// TIA Portal project "izpitni_projekt_v1_final" (V15.1)

(* hardware
DEVICE "S7-1200 station_1"  S7-1200 Station
   slot 0: "Rack_0"  S7-1200 Rack  Rack  V1.0
   slot 1: "PLC_1"  CPU 1214C DC/DC/DC  6ES7 214-1AG40-0XB0  V4.2
   slot 3: "AQ 1x12BIT_1"  AQ1 signal board  6ES7 232-4HA30-0XB0  V1.0
DEVICE "HMI_1"  TP900 Comfort
   slot 0: "HMI_1"  TP900 Comfort  6AV2 124-0JC01-0AX0  15.1.0.0
   slot 1: "HMI_RT_1"  TP900 Comfort  6AV2 124-0JC01-0AX0  15.1.0.0
   slot 5: "HMI_1.IE_CP_1"  PROFINET Interface  15.0.1.0
      slot 1: "PROFINET Interface_1"  PROFINET Interface
         slot 1: "Port_1"  Port
         slot 2: "Port_2"  Port
   slot 7: "HMI_1.MPI/DP_CP_1"  MPI/DP Interface  15.0.1.0
*)

// ===== PLC "PLC_1"  CPU 1214C DC/DC/DC =====
// protected blocks, not shown: "črna_škatlica"

VAR_GLOBAL   // PLC tag table "Default tag table"
   "Tag_1" AT %M0.0 : Bool;
   "Tag_2" AT %M0.1 : Bool;
   "Tag_3" AT %M0.2 : Bool;
   "Clock_Byte" AT %MB0 : Byte;
   "Clock_10Hz" AT %M0.0 : Bool;
   "Clock_5Hz" AT %M0.1 : Bool;
   "Clock_2.5Hz" AT %M0.2 : Bool;
   "Clock_2Hz" AT %M0.3 : Bool;
   "Clock_1.25Hz" AT %M0.4 : Bool;
   "Clock_1Hz" AT %M0.5 : Bool;
   "Clock_0.625Hz" AT %M0.6 : Bool;
   "Clock_0.5Hz" AT %M0.7 : Bool;
END_VAR

DATA_BLOCK "podatki_procesa"   // DB2
{ S7_Optimized_Access := 'TRUE' }
VERSION : 0.1
   VAR
      t_prek : Real := 0.05;   // čas prekinitve v s
      T_A : Real := 40.0;   // temperatura reagenta A
      T_B : Real := 20.0;   // temperatura reagenta B
      T_ok : Real := 20.0;   // temperatura okolice
      T_žel_max : Real := 85.0;   // maksimalna želena temperatura procesa
      deltaT_grad : Real := 1.0;   // gradient spremembe temperature (rampa v st. C/s)
      fi_A_max : Real := 500.0;   // pretok v ml/s
      fi_B_max : Real := 500.0;   // pretok v ml/s
      fi_OUT_max : Real := 500.0;   // pretok v ml/s
      t_heat : Real := 20.0;   // trajanje koraka 3 (vzdrževanje konst. temp.)
      ro_A : Real := 0.81;
      ro_B : Real := 1.0;
      "%_A" : Real := 0.96;
      V_žel : Real;
      "%_žel" : Real;
      T_Žel : Real;
      V_A : Real;
      V_B : Real;
      Grelec1_power : DInt := 5000;
      Grelec2_power : DInt := 20000;
      Grelec3_power : DInt := 70000;
      Spec_Toplota_Voda : Int := 4182;
      Spec_Toplota_Alkohol : Int := 2440;
      Toplotne_Izgube_Koeficient : Real := -2.409683;   // Izmerjene Toplotne izgube 289.0, 267.5585, trial & error -2.409683
      Toplotne_Izgube_Voda : Real := 400.0;   // Somehow so Toplotne izgube povezane z % razkuzila xd
   END_VAR
BEGIN
END_DATA_BLOCK

DATA_BLOCK "spremenljivke"   // DB3
{ S7_Optimized_Access := 'TRUE' }
VERSION : 0.1
   VAR
      reset_DB : Bool;   // tipka reset
      glavno_stikalo_DB : Bool := true;
      zasilni_izklop_DB : Bool;
      avtomatično : Bool := true;
      Ventil_voda : Bool;
      Ventil_alkohol : Bool;
      Ventil_out : Bool;
      Mešalo : Bool;
      Korak1 : Bool;
      Korak2 : Bool;
      Korak3 : Bool;
      Korak4 : Bool;
      Grelec1 : Bool;
      Grelec2 : Bool;
      Grelec3 : Bool;
      Volumen : Real;
      Temperatura : Real;
      prejsna_temp : Real;
      Temp_gradient : Real;
      "%_trenutni" : Real;
      L_zg : Bool;
      L_sp : Bool;
      Pretok_alkohol_mapped : Real;
      Pretok_alkohol : Real;
      Pretok_Voda_mapped : Real;
      Pretok_Voda : Real;
      RMSE_T : Real;
      Error : Word;
   END_VAR
BEGIN
END_DATA_BLOCK

DATA_BLOCK "Korak1_DB"   // DB4
{ S7_Optimized_Access := 'TRUE' }
VERSION : 0.1
// stored: InstanceOfName Korak1
"Korak1"
BEGIN
END_DATA_BLOCK

DATA_BLOCK "Korak3_DB"   // DB5
{ S7_Optimized_Access := 'TRUE' }
VERSION : 0.1
// stored: InstanceOfName Korak3
"Korak3"
BEGIN
END_DATA_BLOCK

DATA_BLOCK "Korak2_DB"   // DB7
{ S7_Optimized_Access := 'TRUE' }
VERSION : 0.1
// stored: InstanceOfName Korak2
"Korak2"
BEGIN
END_DATA_BLOCK

FUNCTION_BLOCK "Korak1"   // FB2, LAD
{ S7_Optimized_Access := 'TRUE' }
VERSION : 0.1
   VAR_INPUT
      reset : Bool;
      "counter" : DInt;
   END_VAR
   VAR_OUTPUT
      finnished : Bool;
   END_VAR
   VAR
      interrupts_count : DInt;
   END_VAR
   VAR_TEMP
      "cas ventil voda" : Time;
      interrupts_voda : Int;
      "cas ventil alkohol" : Time;
      interrupts_alkohol : Int;
   END_VAR
   VAR_TEMP   // added for the SCL form of the ladder/FBD networks
      _w1 : Bool;
      _w2 : Bool;
   END_VAR
BEGIN

REGION Network 1
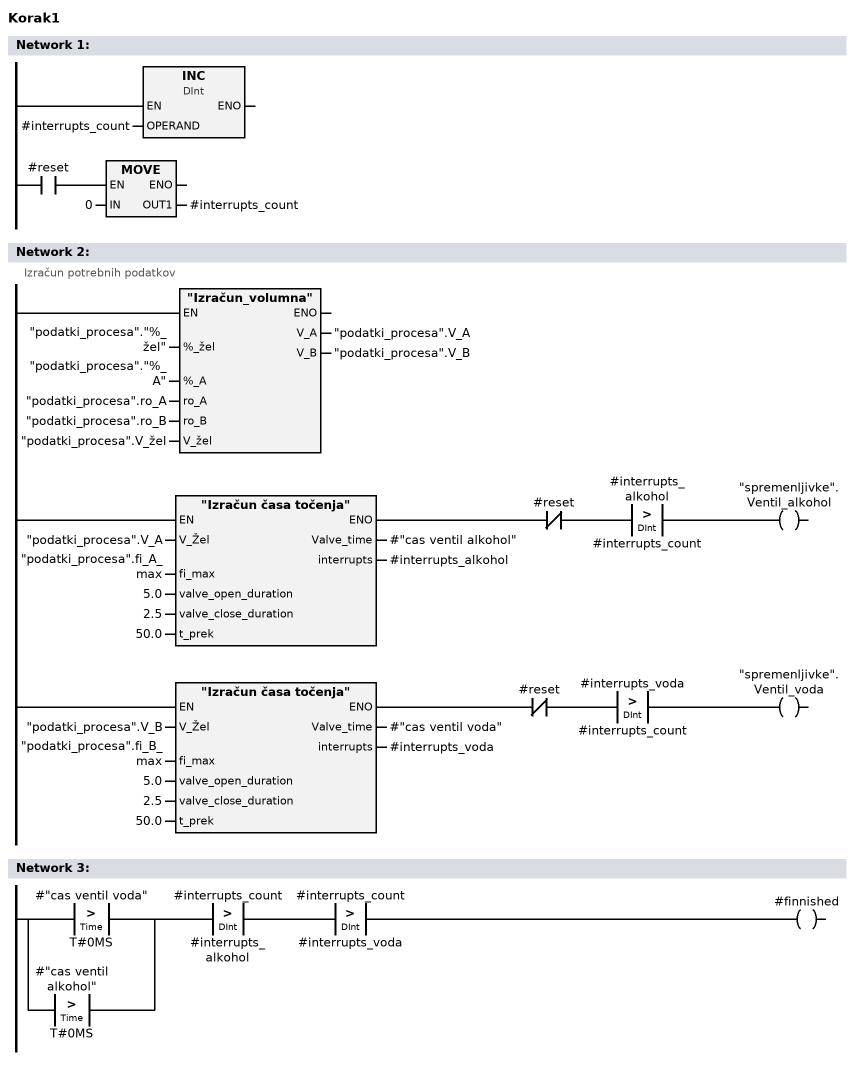
   RUNG wire#powerrail
      { S7_Templates := "DestType := DInt" } Inc( #interrupts_count )
   END_RUNG
   RUNG wire#powerrail
      Contact( #reset )
      Move(in := 0, out1 => #interrupts_count)
   END_RUNG
   // the same network as SCL:
   #interrupts_count := #interrupts_count + 1;
   IF #reset THEN #interrupts_count := 0; END_IF;
END_REGION

REGION Network 2
   // Izračun potrebnih podatkov
   RUNG wire#powerrail
      "Izračun_volumna"("%_žel" := "podatki_procesa"."%_žel", "%_A" := "podatki_procesa"."%_A", ro_A := "podatki_procesa".ro_A, ro_B := "podatki_procesa".ro_B, V_žel := "podatki_procesa".V_žel, V_A => "podatki_procesa".V_A, V_B => "podatki_procesa".V_B)
   END_RUNG
   RUNG wire#powerrail
      "Izračun časa točenja"(V_Žel := "podatki_procesa".V_A, fi_max := "podatki_procesa".fi_A_max, valve_open_duration := 5.0, valve_close_duration := 2.5, t_prek := 50.0, Valve_time => #"cas ventil alkohol", interrupts => #interrupts_alkohol)
      I_Contact( #reset )
      { S7_Templates := "SrcType := DInt" } GT_Contact(in1 := #interrupts_alkohol, in2 := #interrupts_count)
      Coil( "spremenljivke".Ventil_alkohol )
   END_RUNG
   RUNG wire#powerrail
      "Izračun časa točenja"(V_Žel := "podatki_procesa".V_B, fi_max := "podatki_procesa".fi_B_max, valve_open_duration := 5.0, valve_close_duration := 2.5, t_prek := 50.0, Valve_time => #"cas ventil voda", interrupts => #interrupts_voda)
      I_Contact( #reset )
      { S7_Templates := "SrcType := DInt" } GT_Contact(in1 := #interrupts_voda, in2 := #interrupts_count)
      Coil( "spremenljivke".Ventil_voda )
   END_RUNG
   // the same network as SCL:
   "Izračun_volumna"("%_žel" := "podatki_procesa"."%_žel",
                     "%_A" := "podatki_procesa"."%_A",
                     ro_A := "podatki_procesa".ro_A,
                     ro_B := "podatki_procesa".ro_B,
                     V_žel := "podatki_procesa".V_žel,
                     V_A => "podatki_procesa".V_A,
                     V_B => "podatki_procesa".V_B);
   "Izračun časa točenja"(V_Žel := "podatki_procesa".V_A,
                          fi_max := "podatki_procesa".fi_A_max,
                          valve_open_duration := 5.0,
                          valve_close_duration := 2.5,
                          t_prek := 50.0,
                          Valve_time => #"cas ventil alkohol",
                          interrupts => #interrupts_alkohol,
                          ENO => #_w1);
   "spremenljivke".Ventil_alkohol := #_w1 AND NOT #reset AND (#interrupts_alkohol > #interrupts_count);
   "Izračun časa točenja"(V_Žel := "podatki_procesa".V_B,
                          fi_max := "podatki_procesa".fi_B_max,
                          valve_open_duration := 5.0,
                          valve_close_duration := 2.5,
                          t_prek := 50.0,
                          Valve_time => #"cas ventil voda",
                          interrupts => #interrupts_voda,
                          ENO => #_w2);
   "spremenljivke".Ventil_voda := #_w2 AND NOT #reset AND (#interrupts_voda > #interrupts_count);
END_REGION

REGION Network 3
   RUNG wire#powerrail
      { S7_Templates := "SrcType := Time" } GT_Contact(in1 := #"cas ventil voda", in2 := T#0MS)
      wire#w1
      { S7_Templates := "SrcType := DInt" } GT_Contact(in1 := #interrupts_count, in2 := #interrupts_alkohol)
      { S7_Templates := "SrcType := DInt" } GT_Contact(in1 := #interrupts_count, in2 := #interrupts_voda)
      Coil( #finnished )
   END_RUNG
   RUNG wire#powerrail
      { S7_Templates := "SrcType := Time" } GT_Contact(in1 := #"cas ventil alkohol", in2 := T#0MS)
   END_RUNG wire#w1
   // the same network as SCL:
   #finnished := ((#"cas ventil voda" > T#0MS) OR (#"cas ventil alkohol" > T#0MS)) AND (#interrupts_count > #interrupts_alkohol) AND (#interrupts_count > #interrupts_voda);
END_REGION
END_FUNCTION_BLOCK

FUNCTION_BLOCK "Korak2"   // FB3, LAD
{ S7_Optimized_Access := 'TRUE' }
VERSION : 0.1
   VAR_INPUT
      reset : Bool;
   END_VAR
   VAR_OUTPUT
      finnished : Bool;
   END_VAR
   VAR
      interrupts_count : DInt;
      Upravljaj_grelce_Instance : "Upravljaj_grelce";
      Upravljaj_grelce_Instance_1 : "Upravljaj_grelce";
   END_VAR
   VAR_TEMP
      "Energija/K_Total" : Real;
      "Energija/K_Alkohol" : Real;
      "Energija/K_Voda_Alko" : Real;
      "Energija/K_Voda" : Real;
      "%_vode_v_alko" : Real;
      Toplotne_izbuge : Real;
      Potrebna_energija : Real;
      ElapsedTime : Time;
   END_VAR
BEGIN

REGION Network 1
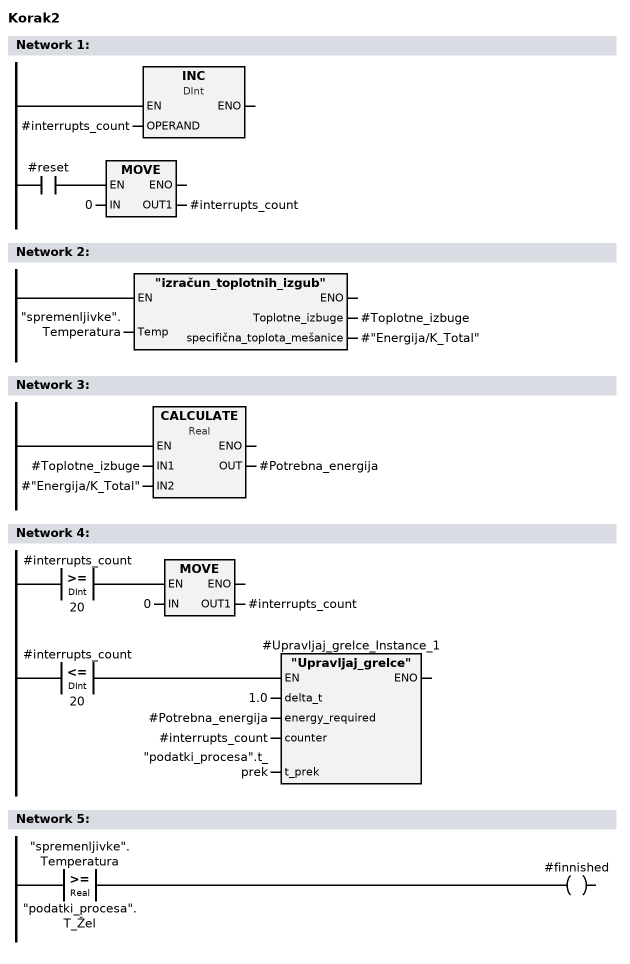
   RUNG wire#powerrail
      { S7_Templates := "DestType := DInt" } Inc( #interrupts_count )
   END_RUNG
   RUNG wire#powerrail
      Contact( #reset )
      Move(in := 0, out1 => #interrupts_count)
   END_RUNG
   // the same network as SCL:
   #interrupts_count := #interrupts_count + 1;
   IF #reset THEN #interrupts_count := 0; END_IF;
END_REGION

REGION Network 2
   RUNG wire#powerrail
      "izračun_toplotnih_izgub"(Temp := "spremenljivke".Temperatura, Toplotne_izbuge => #Toplotne_izbuge, specifična_toplota_mešanice => #"Energija/K_Total")
   END_RUNG
   // the same network as SCL:
   "izračun_toplotnih_izgub"(Temp := "spremenljivke".Temperatura,
                           Toplotne_izbuge => #Toplotne_izbuge,
                           specifična_toplota_mešanice => #"Energija/K_Total");
END_REGION

REGION Network 3
   RUNG wire#powerrail
      { S7_Templates := "SrcType := Real"; S7_Expression := "(IN1 + IN2)" } Calculate(in1 := #Toplotne_izbuge, in2 := #"Energija/K_Total", out => #Potrebna_energija)
   END_RUNG
   // the same network as SCL:
   #Potrebna_energija := (#Toplotne_izbuge + #"Energija/K_Total");
END_REGION

REGION Network 4
   RUNG wire#powerrail
      { S7_Templates := "SrcType := DInt" } GE_Contact(in1 := #interrupts_count, in2 := 20)
      Move(in := 0, out1 => #interrupts_count)
   END_RUNG
   RUNG wire#powerrail
      { S7_Templates := "SrcType := DInt" } LE_Contact(in1 := #interrupts_count, in2 := 20)
      #Upravljaj_grelce_Instance_1(delta_t := 1.0, energy_required := #Potrebna_energija, "counter" := #interrupts_count, t_prek := "podatki_procesa".t_prek)
   END_RUNG
   // the same network as SCL:
   IF #interrupts_count >= 20 THEN #interrupts_count := 0; END_IF;
   IF #interrupts_count <= 20 THEN
       #Upravljaj_grelce_Instance_1(delta_t := 1.0,   // "Upravljaj_grelce"
                               energy_required := #Potrebna_energija,
                               "counter" := #interrupts_count,
                               t_prek := "podatki_procesa".t_prek);
   END_IF;
END_REGION

REGION Network 5
   RUNG wire#powerrail
      { S7_Templates := "SrcType := Real" } GE_Contact(in1 := "spremenljivke".Temperatura, in2 := "podatki_procesa".T_Žel)
      Coil( #finnished )
   END_RUNG
   // the same network as SCL:
   #finnished := "spremenljivke".Temperatura >= "podatki_procesa".T_Žel;
END_REGION
END_FUNCTION_BLOCK

FUNCTION_BLOCK "Upravljaj_grelce"   // FB4, LAD
{ S7_Optimized_Access := 'TRUE' }
VERSION : 0.1
   VAR_INPUT
      delta_t : Real;
      energy_required : LReal;
      "counter" : Int;
      t_prek : Real;
   END_VAR
   VAR
      energy_delivered : LReal;
      energy_missing : Real;
   END_VAR
   VAR_TEMP
      power : Real;
      energy_heater1 : Real;
      energy_heater2 : Real;
      energy_heater3 : Real;
   END_VAR
   VAR_TEMP   // added for the SCL form of the ladder/FBD networks
      _w1 : Bool;
   END_VAR
BEGIN

REGION Network 1
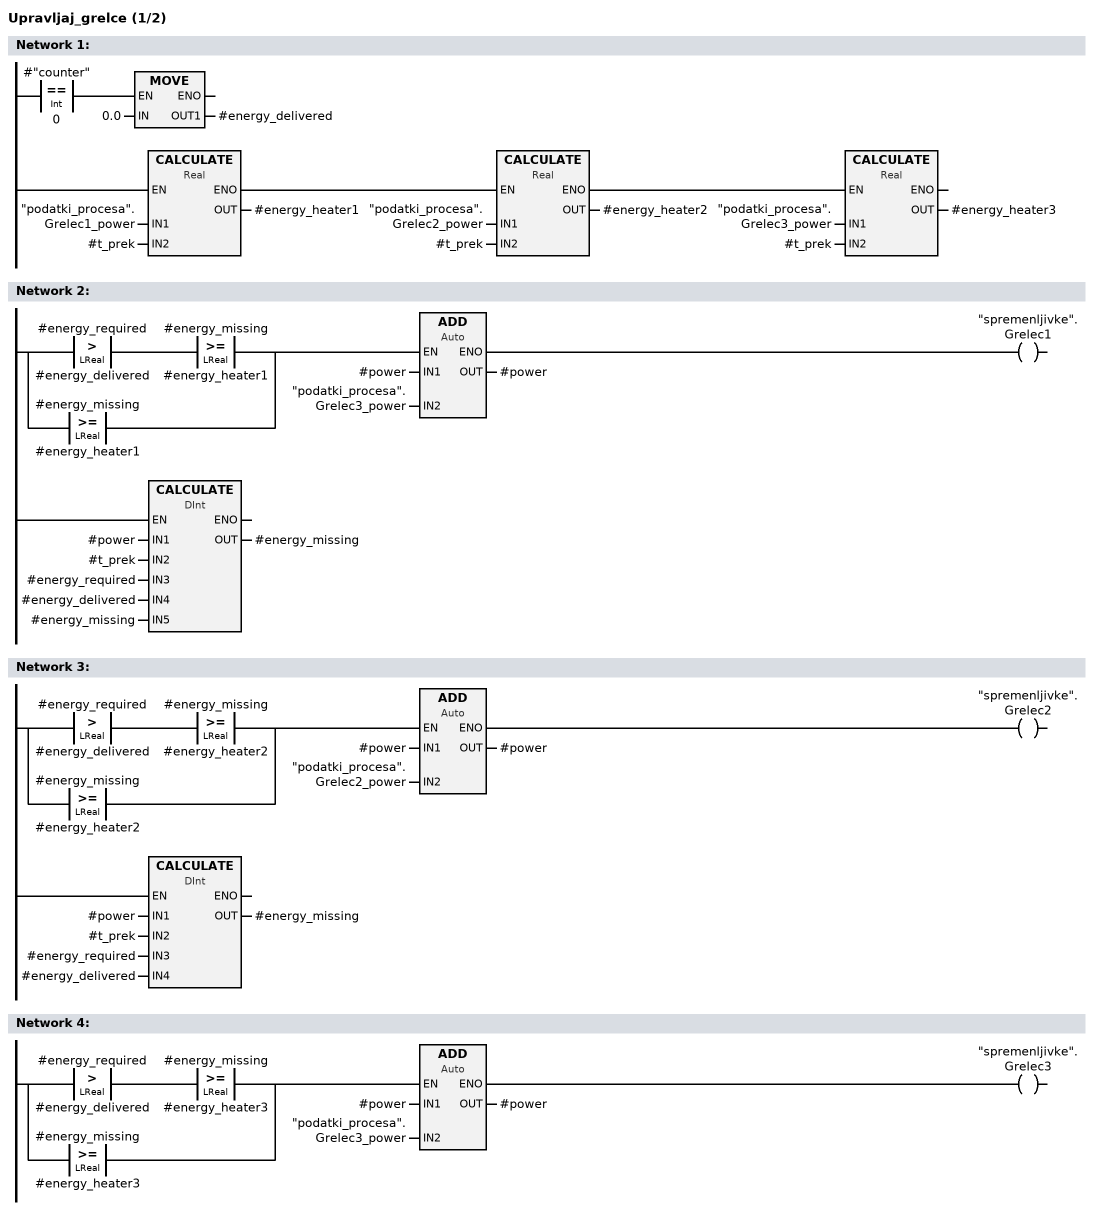
   RUNG wire#powerrail
      { S7_Templates := "SrcType := Int" } EQ_Contact(in1 := #"counter", in2 := 0)
      Move(in := 0.0, out1 => #energy_delivered)
   END_RUNG
   RUNG wire#powerrail
      { S7_Templates := "SrcType := Real"; S7_Expression := "IN1*IN2" } Calculate(in1 := "podatki_procesa".Grelec1_power, in2 := #t_prek, out => #energy_heater1)
      { S7_Templates := "SrcType := Real"; S7_Expression := "IN1*IN2" } Calculate(in1 := "podatki_procesa".Grelec2_power, in2 := #t_prek, out => #energy_heater2)
      { S7_Templates := "SrcType := Real"; S7_Expression := "IN1*IN2" } Calculate(in1 := "podatki_procesa".Grelec3_power, in2 := #t_prek, out => #energy_heater3)
   END_RUNG
   // the same network as SCL:
   IF #"counter" = 0 THEN #energy_delivered := 0.0; END_IF;
   #energy_heater1 := "podatki_procesa".Grelec1_power*#t_prek;
   #energy_heater2 := "podatki_procesa".Grelec2_power*#t_prek;
   #energy_heater3 := "podatki_procesa".Grelec3_power*#t_prek;
END_REGION

REGION Network 2
   RUNG wire#powerrail
      { S7_Templates := "SrcType := LReal" } GT_Contact(in1 := #energy_required, in2 := #energy_delivered)
      { S7_Templates := "SrcType := LReal" } GE_Contact(in1 := #energy_missing, in2 := #energy_heater1)
      wire#w1
      Add(in1 := #power, in2 := "podatki_procesa".Grelec3_power, out => #power)
      Coil( "spremenljivke".Grelec1 )
   END_RUNG
   RUNG wire#powerrail
      { S7_Templates := "SrcType := LReal" } GE_Contact(in1 := #energy_missing, in2 := #energy_heater1)
   END_RUNG wire#w1
   RUNG wire#powerrail
      { S7_Templates := "SrcType := DInt"; S7_Expression := "(IN3-IN4-IN1*IN2 )+ IN5" } Calculate(in1 := #power, in2 := #t_prek, in3 := #energy_required, in4 := #energy_delivered, in5 := #energy_missing, out => #energy_missing)
   END_RUNG
   // the same network as SCL:
   #_w1 := ((#energy_required > #energy_delivered) AND (#energy_missing >= #energy_heater1)) OR (#energy_missing >= #energy_heater1);
   IF #_w1 THEN #power := #power + "podatki_procesa".Grelec3_power; END_IF;
   "spremenljivke".Grelec1 := #_w1;
   #energy_missing := (#energy_required-#energy_delivered-#power*#t_prek )+ #energy_missing;
END_REGION

REGION Network 3
   RUNG wire#powerrail
      { S7_Templates := "SrcType := LReal" } GT_Contact(in1 := #energy_required, in2 := #energy_delivered)
      { S7_Templates := "SrcType := LReal" } GE_Contact(in1 := #energy_missing, in2 := #energy_heater2)
      wire#w1
      Add(in1 := #power, in2 := "podatki_procesa".Grelec2_power, out => #power)
      Coil( "spremenljivke".Grelec2 )
   END_RUNG
   RUNG wire#powerrail
      { S7_Templates := "SrcType := LReal" } GE_Contact(in1 := #energy_missing, in2 := #energy_heater2)
   END_RUNG wire#w1
   RUNG wire#powerrail
      { S7_Templates := "SrcType := DInt"; S7_Expression := "IN3-IN4-IN1*IN2" } Calculate(in1 := #power, in2 := #t_prek, in3 := #energy_required, in4 := #energy_delivered, out => #energy_missing)
   END_RUNG
   // the same network as SCL:
   #_w1 := ((#energy_required > #energy_delivered) AND (#energy_missing >= #energy_heater2)) OR (#energy_missing >= #energy_heater2);
   IF #_w1 THEN #power := #power + "podatki_procesa".Grelec2_power; END_IF;
   "spremenljivke".Grelec2 := #_w1;
   #energy_missing := #energy_required-#energy_delivered-#power*#t_prek;
END_REGION

REGION Network 4
   RUNG wire#powerrail
      { S7_Templates := "SrcType := LReal" } GT_Contact(in1 := #energy_required, in2 := #energy_delivered)
      { S7_Templates := "SrcType := LReal" } GE_Contact(in1 := #energy_missing, in2 := #energy_heater3)
      wire#w1
      Add(in1 := #power, in2 := "podatki_procesa".Grelec3_power, out => #power)
      Coil( "spremenljivke".Grelec3 )
   END_RUNG
   RUNG wire#powerrail
      { S7_Templates := "SrcType := LReal" } GE_Contact(in1 := #energy_missing, in2 := #energy_heater3)
   END_RUNG wire#w1
   // the same network as SCL:
   #_w1 := ((#energy_required > #energy_delivered) AND (#energy_missing >= #energy_heater3)) OR (#energy_missing >= #energy_heater3);
   IF #_w1 THEN #power := #power + "podatki_procesa".Grelec3_power; END_IF;
   "spremenljivke".Grelec3 := #_w1;
END_REGION

REGION Network 5
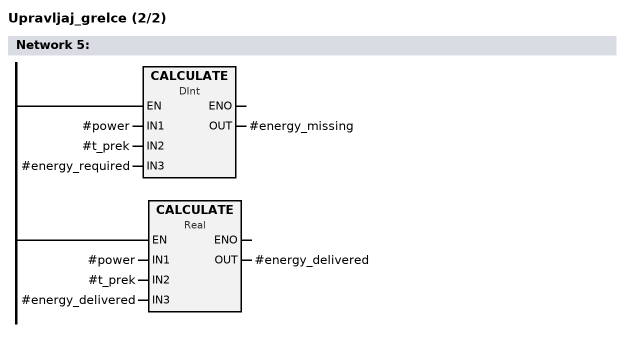
   RUNG wire#powerrail
      { S7_Templates := "SrcType := DInt"; S7_Expression := "IN3-IN1*IN2" } Calculate(in1 := #power, in2 := #t_prek, in3 := #energy_required, out => #energy_missing)
   END_RUNG
   RUNG wire#powerrail
      { S7_Templates := "SrcType := Real"; S7_Expression := "IN3 + IN1 * IN2" } Calculate(in1 := #power, in2 := #t_prek, in3 := #energy_delivered, out => #energy_delivered)
   END_RUNG
   // the same network as SCL:
   #energy_missing := #energy_required-#power*#t_prek;
   #energy_delivered := #energy_delivered + #power * #t_prek;
END_REGION
END_FUNCTION_BLOCK

FUNCTION_BLOCK "Korak3"   // FB5, LAD
{ S7_Optimized_Access := 'TRUE' }
VERSION : 0.1
   VAR_INPUT
      reset : Bool;
   END_VAR
   VAR_OUTPUT
      finnished_1 : Bool;
   END_VAR
   VAR
      Upravljaj_grelce_Instance : "Upravljaj_grelce";
      interrupts_count : DInt;
   END_VAR
   VAR_TEMP
      "toplotne izgube" : Real;
      "specificna toplota" : Real;
   END_VAR
BEGIN

REGION Network 1
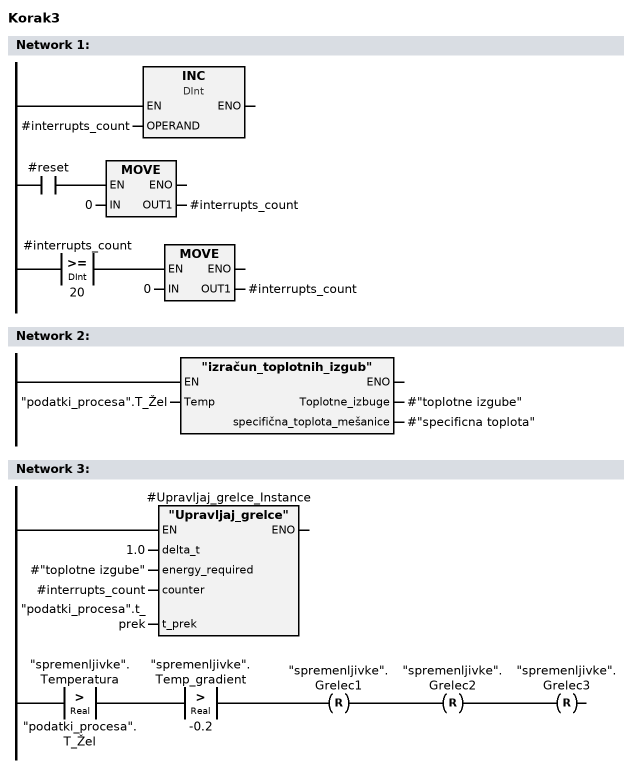
   RUNG wire#powerrail
      { S7_Templates := "DestType := DInt" } Inc( #interrupts_count )
   END_RUNG
   RUNG wire#powerrail
      Contact( #reset )
      Move(in := 0, out1 => #interrupts_count)
   END_RUNG
   RUNG wire#powerrail
      { S7_Templates := "SrcType := DInt" } GE_Contact(in1 := #interrupts_count, in2 := 20)
      Move(in := 0, out1 => #interrupts_count)
   END_RUNG
   // the same network as SCL:
   #interrupts_count := #interrupts_count + 1;
   IF #reset THEN #interrupts_count := 0; END_IF;
   IF #interrupts_count >= 20 THEN #interrupts_count := 0; END_IF;
END_REGION

REGION Network 2
   RUNG wire#powerrail
      "izračun_toplotnih_izgub"(Temp := "podatki_procesa".T_Žel, Toplotne_izbuge => #"toplotne izgube", specifična_toplota_mešanice => #"specificna toplota")
   END_RUNG
   // the same network as SCL:
   "izračun_toplotnih_izgub"(Temp := "podatki_procesa".T_Žel,
                           Toplotne_izbuge => #"toplotne izgube",
                           specifična_toplota_mešanice => #"specificna toplota");
END_REGION

REGION Network 3
   RUNG wire#powerrail
      #Upravljaj_grelce_Instance(delta_t := 1.0, energy_required := #"toplotne izgube", "counter" := #interrupts_count, t_prek := "podatki_procesa".t_prek)
   END_RUNG
   RUNG wire#powerrail
      { S7_Templates := "SrcType := Real" } GT_Contact(in1 := "spremenljivke".Temperatura, in2 := "podatki_procesa".T_Žel)
      { S7_Templates := "SrcType := Real" } GT_Contact(in1 := "spremenljivke".Temp_gradient, in2 := -0.2)
      R_Coil( "spremenljivke".Grelec1 )
      R_Coil( "spremenljivke".Grelec2 )
      R_Coil( "spremenljivke".Grelec3 )
   END_RUNG
   // the same network as SCL:
   #Upravljaj_grelce_Instance(delta_t := 1.0,   // "Upravljaj_grelce"
                           energy_required := #"toplotne izgube",
                           "counter" := #interrupts_count,
                           t_prek := "podatki_procesa".t_prek);
   IF ("spremenljivke".Temperatura > "podatki_procesa".T_Žel) AND ("spremenljivke".Temp_gradient > (-0.2)) THEN
       "spremenljivke".Grelec1 := FALSE;
       "spremenljivke".Grelec2 := FALSE;
       "spremenljivke".Grelec3 := FALSE;
   END_IF;
END_REGION
END_FUNCTION_BLOCK

FUNCTION "map_Flow_Sensor" : Void   // FC1, LAD
{ S7_Optimized_Access := 'TRUE' }
VERSION : 0.1
   VAR_INPUT
      input_value : Real;
      max_value : Real;
   END_VAR
   VAR_OUTPUT
      output_value : Real;
   END_VAR
   VAR_TEMP
      norm_Value : Real;
   END_VAR
BEGIN

REGION Network 1
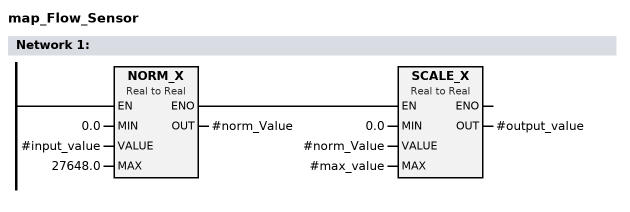
   RUNG wire#powerrail
      { S7_Templates := "[SrcType := Real, DestType := Real]" } Normalize(min := 0.0, value := #input_value, max := 27648.0, out => #norm_Value)
      { S7_Templates := "[SrcType := Real, DestType := Real]" } Scale(min := 0.0, value := #norm_Value, max := #max_value, out => #output_value)
   END_RUNG
   // the same network as SCL:
   #norm_Value := NORM_X(MIN := 0.0, VALUE := #input_value, MAX := 27648.0);
   #output_value := SCALE_X(MIN := 0.0, VALUE := #norm_Value, MAX := #max_value);
END_REGION
END_FUNCTION

FUNCTION "Izračun_volumna" : Void   // FC2, LAD
{ S7_Optimized_Access := 'TRUE' }
VERSION : 0.1
   VAR_INPUT
      "%_žel" : Real;
      "%_A" : Real;
      ro_A : Real;
      ro_B : Real;
      V_žel : Real;
   END_VAR
   VAR_OUTPUT
      V_A : Real;
      V_B : Real;
   END_VAR
   VAR_TEMP
      "V_B/V_A" : Real;   // Razmerje volumen Vode / Volumen Alkohola
   END_VAR
BEGIN

REGION Network 1
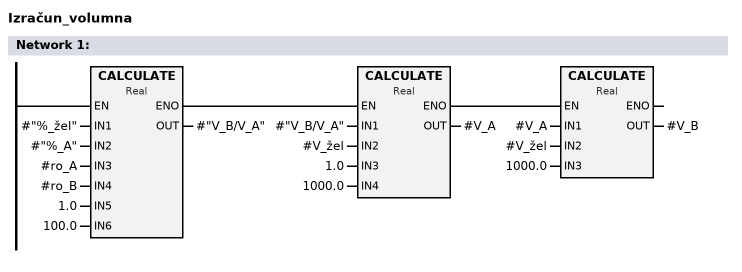
   RUNG wire#powerrail
      { S7_Templates := "SrcType := Real"; S7_Expression := "((IN3 * IN2)/((IN1/IN6) * IN4)) - ((IN3*(IN5-IN2))/IN4) -((IN3 * IN2)/(IN4))" } Calculate(in1 := #"%_žel", in2 := #"%_A", in3 := #ro_A, in4 := #ro_B, in5 := 1.0, in6 := 100.0, out => #"V_B/V_A")
      { S7_Templates := "SrcType := Real"; S7_Expression := "(IN2*IN4)/(IN3+IN1)" } Calculate(in1 := #"V_B/V_A", in2 := #V_žel, in3 := 1.0, in4 := 1000.0, out => #V_A)
      { S7_Templates := "SrcType := Real"; S7_Expression := "(IN2 * IN3) - IN1" } Calculate(in1 := #V_A, in2 := #V_žel, in3 := 1000.0, out => #V_B)
   END_RUNG
   // the same network as SCL:
   #"V_B/V_A" := ((#ro_A * #"%_A")/((#"%_žel"/100.0) * #ro_B)) - ((#ro_A*(1.0-#"%_A"))/#ro_B) -((#ro_A * #"%_A")/(#ro_B));
   #V_A := (#V_žel*1000.0)/(1.0+#"V_B/V_A");
   #V_B := (#V_žel * 1000.0) - #V_A;
END_REGION
END_FUNCTION

FUNCTION "izračun_toplotnih_izgub" : Void   // FC3, LAD
{ S7_Optimized_Access := 'TRUE' }
VERSION : 0.1
   VAR_INPUT
      Temp : Real;
   END_VAR
   VAR_OUTPUT
      Toplotne_izbuge : Real;
      specifična_toplota_mešanice : Real;
   END_VAR
   VAR_TEMP
      "Energija/K_Alkohol" : Real;
      "Energija/K_Voda_Alko" : Real;
      "Energija/K_Voda" : Real;
      "%_vode_v_alko" : Real;
      Potrebna_energija : Real;
   END_VAR
   VAR_TEMP   // added for the SCL form of the ladder/FBD networks
      _w1 : Bool;
   END_VAR
BEGIN

REGION Network 1
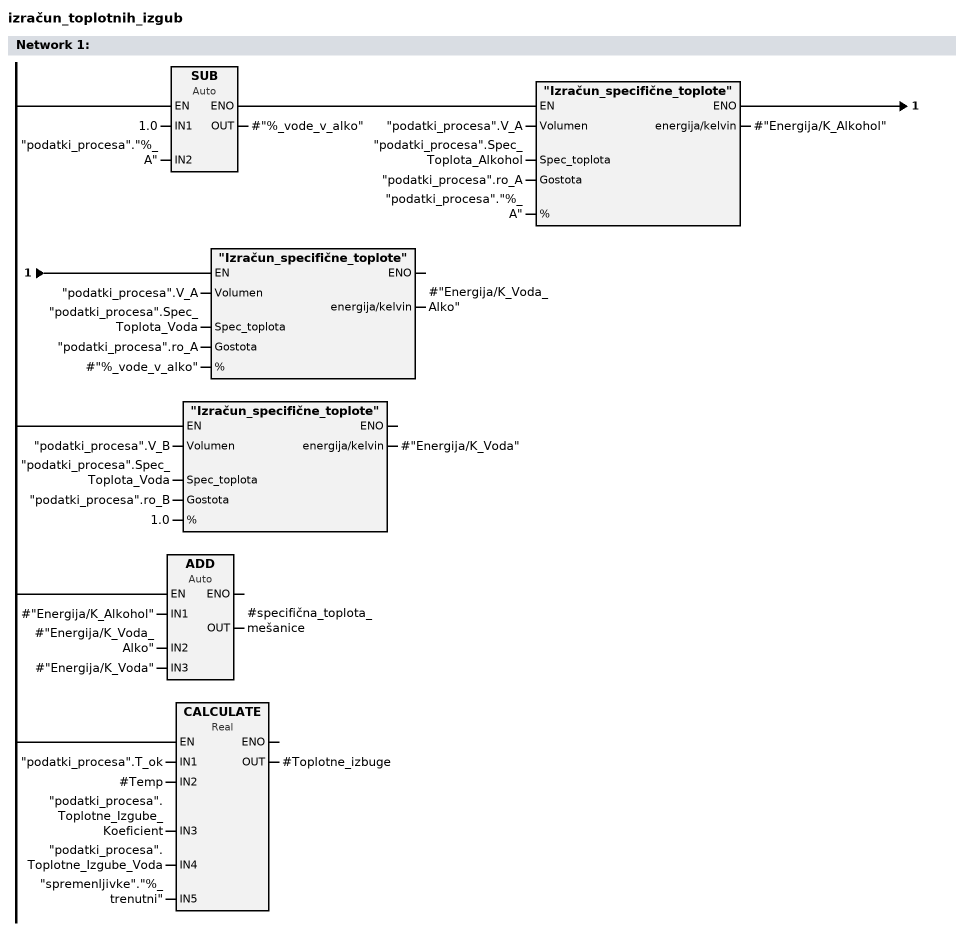
   RUNG wire#powerrail
      Sub(in1 := 1.0, in2 := "podatki_procesa"."%_A", out => #"%_vode_v_alko")
      "Izračun_specifične_toplote"(Volumen := "podatki_procesa".V_A, Spec_toplota := "podatki_procesa".Spec_Toplota_Alkohol, Gostota := "podatki_procesa".ro_A, "%" := "podatki_procesa"."%_A", "energija/kelvin" => #"Energija/K_Alkohol")
      "Izračun_specifične_toplote"(Volumen := "podatki_procesa".V_A, Spec_toplota := "podatki_procesa".Spec_Toplota_Voda, Gostota := "podatki_procesa".ro_A, "%" := #"%_vode_v_alko", "energija/kelvin" => #"Energija/K_Voda_Alko")
   END_RUNG
   RUNG wire#powerrail
      "Izračun_specifične_toplote"(Volumen := "podatki_procesa".V_B, Spec_toplota := "podatki_procesa".Spec_Toplota_Voda, Gostota := "podatki_procesa".ro_B, "%" := 1.0, "energija/kelvin" => #"Energija/K_Voda")
   END_RUNG
   RUNG wire#powerrail
      Add(in1 := #"Energija/K_Alkohol", in2 := #"Energija/K_Voda_Alko", in3 := #"Energija/K_Voda", out => #specifična_toplota_mešanice)
   END_RUNG
   RUNG wire#powerrail
      { S7_Templates := "SrcType := Real"; S7_Expression := "(IN3*IN5 + IN4) * (IN2-IN1)" } Calculate(in1 := "podatki_procesa".T_ok, in2 := #Temp, in3 := "podatki_procesa".Toplotne_Izgube_Koeficient, in4 := "podatki_procesa".Toplotne_Izgube_Voda, in5 := "spremenljivke"."%_trenutni", out => #Toplotne_izbuge)
   END_RUNG
   // the same network as SCL:
   #"%_vode_v_alko" := 1.0 - "podatki_procesa"."%_A";
   "Izračun_specifične_toplote"(Volumen := "podatki_procesa".V_A,
                           Spec_toplota := "podatki_procesa".Spec_Toplota_Alkohol,
                           Gostota := "podatki_procesa".ro_A,
                           "%" := "podatki_procesa"."%_A",
                           "energija/kelvin" => #"Energija/K_Alkohol",
                           ENO => #_w1);
   IF #_w1 THEN
       "Izračun_specifične_toplote"(Volumen := "podatki_procesa".V_A,
                               Spec_toplota := "podatki_procesa".Spec_Toplota_Voda,
                               Gostota := "podatki_procesa".ro_A,
                               "%" := #"%_vode_v_alko",
                               "energija/kelvin" => #"Energija/K_Voda_Alko");
   END_IF;
   "Izračun_specifične_toplote"(Volumen := "podatki_procesa".V_B,
                           Spec_toplota := "podatki_procesa".Spec_Toplota_Voda,
                           Gostota := "podatki_procesa".ro_B,
                           "%" := 1.0,
                           "energija/kelvin" => #"Energija/K_Voda");
   #specifična_toplota_mešanice := #"Energija/K_Alkohol" + #"Energija/K_Voda_Alko" + #"Energija/K_Voda";
   #Toplotne_izbuge := ("podatki_procesa".Toplotne_Izgube_Koeficient*"spremenljivke"."%_trenutni" + "podatki_procesa".Toplotne_Izgube_Voda) * (#Temp-"podatki_procesa".T_ok);
END_REGION
END_FUNCTION

FUNCTION "Izračun časa točenja" : Void   // FC4, LAD
{ S7_Optimized_Access := 'TRUE' }
VERSION : 0.1
   VAR_INPUT
      V_Žel : Real;
      fi_max : Real;
      valve_open_duration : Real;
      valve_close_duration : Real;
      t_prek : Real;
   END_VAR
   VAR_OUTPUT
      Valve_time : Time;
      interrupts : Int;
   END_VAR
   VAR_TEMP
      opening_volume_flown : Real;
      opening_coeficient : Real;
      closing_volume_flown : Real;
      closing_coeficient : Real;
      valve_total_volume_flown : Real;
      "e" : Bool;
      Valve_time_real : Int;
   END_VAR
BEGIN

REGION Network 1
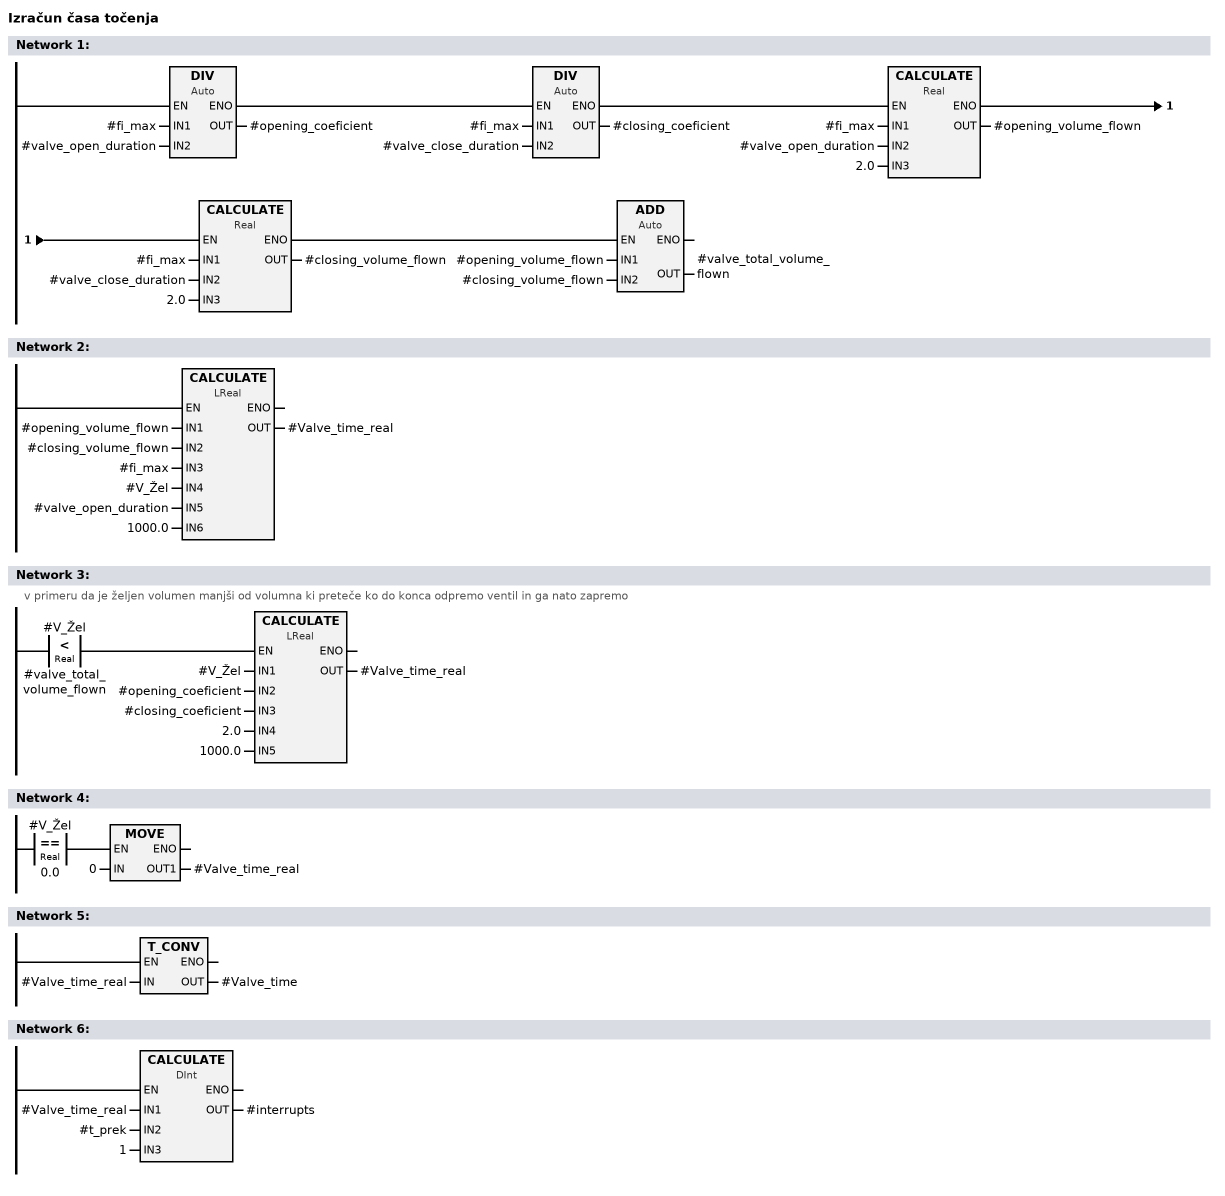
   RUNG wire#powerrail
      Div(in1 := #fi_max, in2 := #valve_open_duration, out => #opening_coeficient)
      Div(in1 := #fi_max, in2 := #valve_close_duration, out => #closing_coeficient)
      { S7_Templates := "SrcType := Real"; S7_Expression := "IN1*IN2/IN3" } Calculate(in1 := #fi_max, in2 := #valve_open_duration, in3 := 2.0, out => #opening_volume_flown)
      { S7_Templates := "SrcType := Real"; S7_Expression := "IN1*IN2/IN3" } Calculate(in1 := #fi_max, in2 := #valve_close_duration, in3 := 2.0, out => #closing_volume_flown)
      Add(in1 := #opening_volume_flown, in2 := #closing_volume_flown, out => #valve_total_volume_flown)
   END_RUNG
   // the same network as SCL:
   #opening_coeficient := #fi_max / #valve_open_duration;
   #closing_coeficient := #fi_max / #valve_close_duration;
   #opening_volume_flown := #fi_max*#valve_open_duration/2.0;
   #closing_volume_flown := #fi_max*#valve_close_duration/2.0;
   #valve_total_volume_flown := #opening_volume_flown + #closing_volume_flown;
END_REGION

REGION Network 2
   RUNG wire#powerrail
      { S7_Templates := "SrcType := LReal"; S7_Expression := "((IN4-IN1-IN2)/(IN3) + IN5)*IN6" } Calculate(in1 := #opening_volume_flown, in2 := #closing_volume_flown, in3 := #fi_max, in4 := #V_Žel, in5 := #valve_open_duration, in6 := 1000.0, out => #Valve_time_real)
   END_RUNG
   // the same network as SCL:
   #Valve_time_real := ((#V_Žel-#opening_volume_flown-#closing_volume_flown)/(#fi_max) + #valve_open_duration)*1000.0;
END_REGION

REGION Network 3
   // v primeru da je željen volumen manjši od volumna ki preteče ko do konca odpremo ventil in ga nato zapremo
   RUNG wire#powerrail
      { S7_Templates := "SrcType := Real" } LT_Contact(in1 := #V_Žel, in2 := #valve_total_volume_flown)
      { S7_Templates := "SrcType := LReal"; S7_Expression := "SQRT(IN1/((IN2/IN4)+(IN2*IN2/IN3)))*IN5" } Calculate(in1 := #V_Žel, in2 := #opening_coeficient, in3 := #closing_coeficient, in4 := 2.0, in5 := 1000.0, out => #Valve_time_real)
   END_RUNG
   // the same network as SCL:
   IF #V_Žel < #valve_total_volume_flown THEN
       #Valve_time_real := SQRT(#V_Žel/((#opening_coeficient/2.0)+(#opening_coeficient*#opening_coeficient/#closing_coeficient)))*1000.0;
   END_IF;
END_REGION

REGION Network 4
   RUNG wire#powerrail
      { S7_Templates := "SrcType := Real" } EQ_Contact(in1 := #V_Žel, in2 := 0.0)
      Move(in := 0, out1 => #Valve_time_real)
   END_RUNG
   // the same network as SCL:
   IF #V_Žel = 0.0 THEN #Valve_time_real := 0; END_IF;
END_REGION

REGION Network 5
   #Valve_time := T_CONV(IN := #Valve_time_real);
END_REGION

REGION Network 6
   RUNG wire#powerrail
      { S7_Templates := "SrcType := DInt"; S7_Expression := "IN1/IN2 + IN3" } Calculate(in1 := #Valve_time_real, in2 := #t_prek, in3 := 1, out => #interrupts)
   END_RUNG
   // the same network as SCL:
   #interrupts := #Valve_time_real/#t_prek + 1;
END_REGION
END_FUNCTION

FUNCTION "Izračun_specifične_toplote" : Void   // FC5, LAD
{ S7_Optimized_Access := 'TRUE' }
VERSION : 0.1
   VAR_INPUT
      Volumen : Real;
      Spec_toplota : Real;
      Gostota : Real;
      "%" : Real;
   END_VAR
   VAR_OUTPUT
      "energija/kelvin" : LReal;
   END_VAR
BEGIN

REGION Network 1
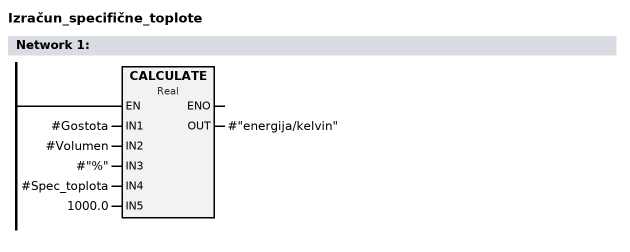
   RUNG wire#powerrail
      { S7_Templates := "SrcType := Real"; S7_Expression := "IN1 * IN2 *IN3 * IN4 / IN5" } Calculate(in1 := #Gostota, in2 := #Volumen, in3 := #"%", in4 := #Spec_toplota, in5 := 1000.0, out => #"energija/kelvin")
   END_RUNG
   // the same network as SCL:
   #"energija/kelvin" := #Gostota * #Volumen *#"%" * #Spec_toplota / 1000.0;
END_REGION
END_FUNCTION

ORGANIZATION_BLOCK "Main"   // OB1, LAD, ProgramCycle
TITLE = "Main Program Sweep (Cycle)"
{ S7_Optimized_Access := 'TRUE' }
VERSION : 0.1
   VAR_INPUT
      Initial_Call : Bool;   // Initial call of this OB
      Remanence : Bool;   // =True, if remanent data are available
   END_VAR
BEGIN
END_ORGANIZATION_BLOCK

ORGANIZATION_BLOCK "Cyclic interrupt"   // OB30, LAD, CyclicInterrupt
{ S7_Optimized_Access := 'TRUE' }
VERSION : 0.1
   VAR_INPUT
      Initial_Call : Bool;   // Initial call of this OB
      Event_Count : Int;   // Events discarded
   END_VAR
   VAR_TEMP
      korak1_finnished : Bool;
      korak2_finnished : Bool;
      korak3_finnished : Bool;
   END_VAR
   VAR CONSTANT
      tempyacetek : Real := 50.0;
   END_VAR
BEGIN

REGION Network 1
   // Mapping pretoka
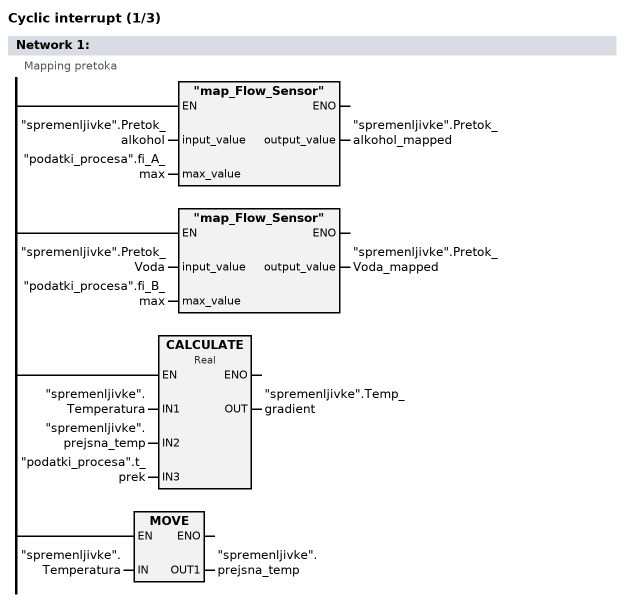
   RUNG wire#powerrail
      "map_Flow_Sensor"(input_value := "spremenljivke".Pretok_alkohol, max_value := "podatki_procesa".fi_A_max, output_value => "spremenljivke".Pretok_alkohol_mapped)
   END_RUNG
   RUNG wire#powerrail
      "map_Flow_Sensor"(input_value := "spremenljivke".Pretok_Voda, max_value := "podatki_procesa".fi_B_max, output_value => "spremenljivke".Pretok_Voda_mapped)
   END_RUNG
   RUNG wire#powerrail
      { S7_Templates := "SrcType := Real"; S7_Expression := "(IN1-IN2)/IN3" } Calculate(in1 := "spremenljivke".Temperatura, in2 := "spremenljivke".prejsna_temp, in3 := "podatki_procesa".t_prek, out => "spremenljivke".Temp_gradient)
   END_RUNG
   RUNG wire#powerrail
      Move(in := "spremenljivke".Temperatura, out1 => "spremenljivke".prejsna_temp)
   END_RUNG
   // the same network as SCL:
   "map_Flow_Sensor"(input_value := "spremenljivke".Pretok_alkohol,
                     max_value := "podatki_procesa".fi_A_max,
                     output_value => "spremenljivke".Pretok_alkohol_mapped);
   "map_Flow_Sensor"(input_value := "spremenljivke".Pretok_Voda,
                     max_value := "podatki_procesa".fi_B_max,
                     output_value => "spremenljivke".Pretok_Voda_mapped);
   "spremenljivke".Temp_gradient := ("spremenljivke".Temperatura-"spremenljivke".prejsna_temp)/"podatki_procesa".t_prek;
   "spremenljivke".prejsna_temp := "spremenljivke".Temperatura;
END_REGION

REGION Network 2
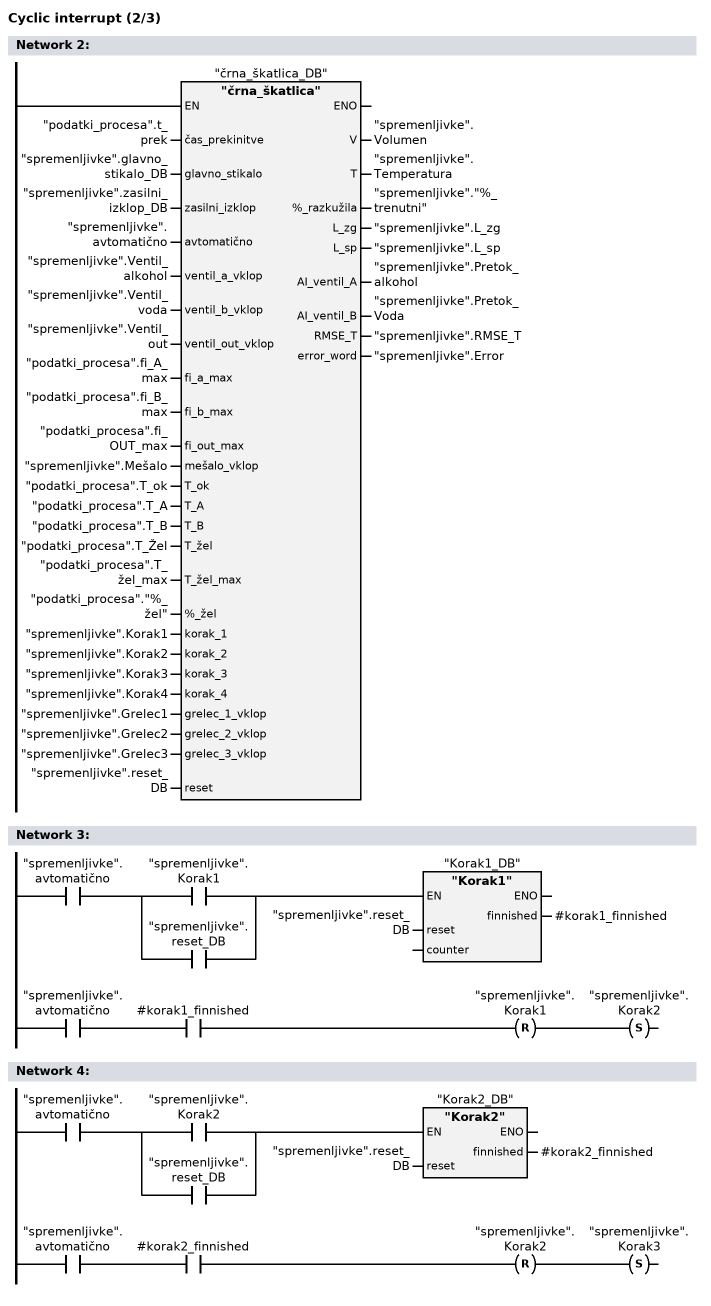
   RUNG wire#powerrail
      "črna_škatlica_DB"(čas_prekinitve := "podatki_procesa".t_prek, glavno_stikalo := "spremenljivke".glavno_stikalo_DB, zasilni_izklop := "spremenljivke".zasilni_izklop_DB, avtomatično := "spremenljivke".avtomatično, ventil_a_vklop := "spremenljivke".Ventil_alkohol, ventil_b_vklop := "spremenljivke".Ventil_voda, ventil_out_vklop := "spremenljivke".Ventil_out, fi_a_max := "podatki_procesa".fi_A_max, fi_b_max := "podatki_procesa".fi_B_max, fi_out_max := "podatki_procesa".fi_OUT_max, mešalo_vklop := "spremenljivke".Mešalo, T_ok := "podatki_procesa".T_ok, T_A := "podatki_procesa".T_A, T_B := "podatki_procesa".T_B, T_žel := "podatki_procesa".T_Žel, T_žel_max := "podatki_procesa".T_žel_max, "%_žel" := "podatki_procesa"."%_žel", korak_1 := "spremenljivke".Korak1, korak_2 := "spremenljivke".Korak2, korak_3 := "spremenljivke".Korak3, korak_4 := "spremenljivke".Korak4, grelec_1_vklop := "spremenljivke".Grelec1, grelec_2_vklop := "spremenljivke".Grelec2, grelec_3_vklop := "spremenljivke".Grelec3, reset := "spremenljivke".reset_DB, V => "spremenljivke".Volumen, T => "spremenljivke".Temperatura, "%_razkužila" => "spremenljivke"."%_trenutni", L_zg => "spremenljivke".L_zg, L_sp => "spremenljivke".L_sp, AI_ventil_A => "spremenljivke".Pretok_alkohol, AI_ventil_B => "spremenljivke".Pretok_Voda, RMSE_T => "spremenljivke".RMSE_T, error_word => "spremenljivke".Error)
   END_RUNG
   // the same network as SCL:
   "črna_škatlica_DB"(čas_prekinitve := "podatki_procesa".t_prek,   // "črna_škatlica"
                      glavno_stikalo := "spremenljivke".glavno_stikalo_DB,
                      zasilni_izklop := "spremenljivke".zasilni_izklop_DB,
                      avtomatično := "spremenljivke".avtomatično,
                      ventil_a_vklop := "spremenljivke".Ventil_alkohol,
                      ventil_b_vklop := "spremenljivke".Ventil_voda,
                      ventil_out_vklop := "spremenljivke".Ventil_out,
                      fi_a_max := "podatki_procesa".fi_A_max,
                      fi_b_max := "podatki_procesa".fi_B_max,
                      fi_out_max := "podatki_procesa".fi_OUT_max,
                      mešalo_vklop := "spremenljivke".Mešalo,
                      T_ok := "podatki_procesa".T_ok,
                      T_A := "podatki_procesa".T_A,
                      T_B := "podatki_procesa".T_B,
                      T_žel := "podatki_procesa".T_Žel,
                      T_žel_max := "podatki_procesa".T_žel_max,
                      "%_žel" := "podatki_procesa"."%_žel",
                      korak_1 := "spremenljivke".Korak1,
                      korak_2 := "spremenljivke".Korak2,
                      korak_3 := "spremenljivke".Korak3,
                      korak_4 := "spremenljivke".Korak4,
                      grelec_1_vklop := "spremenljivke".Grelec1,
                      grelec_2_vklop := "spremenljivke".Grelec2,
                      grelec_3_vklop := "spremenljivke".Grelec3,
                      reset := "spremenljivke".reset_DB,
                      V => "spremenljivke".Volumen,
                      T => "spremenljivke".Temperatura,
                      "%_razkužila" => "spremenljivke"."%_trenutni",
                      L_zg => "spremenljivke".L_zg,
                      L_sp => "spremenljivke".L_sp,
                      AI_ventil_A => "spremenljivke".Pretok_alkohol,
                      AI_ventil_B => "spremenljivke".Pretok_Voda,
                      RMSE_T => "spremenljivke".RMSE_T,
                      error_word => "spremenljivke".Error);
END_REGION

REGION Network 3
   RUNG wire#powerrail
      Contact( "spremenljivke".avtomatično )
      wire#w1
      Contact( "spremenljivke".Korak1 )
      wire#w2
      "Korak1_DB"(reset := "spremenljivke".reset_DB, "counter" :=, finnished => #korak1_finnished)
   END_RUNG
   RUNG wire#w1
      Contact( "spremenljivke".reset_DB )
   END_RUNG wire#w2
   RUNG wire#powerrail
      Contact( "spremenljivke".avtomatično )
      Contact( #korak1_finnished )
      R_Coil( "spremenljivke".Korak1 )
      S_Coil( "spremenljivke".Korak2 )
   END_RUNG
   // the same network as SCL:
   IF "spremenljivke".avtomatično AND ("spremenljivke".Korak1 OR "spremenljivke".reset_DB) THEN
       "Korak1_DB"(reset := "spremenljivke".reset_DB, finnished => #korak1_finnished);   // "Korak1"
   END_IF;
   IF "spremenljivke".avtomatično AND #korak1_finnished THEN
       "spremenljivke".Korak1 := FALSE;
       "spremenljivke".Korak2 := TRUE;
   END_IF;
END_REGION

REGION Network 4
   RUNG wire#powerrail
      Contact( "spremenljivke".avtomatično )
      wire#w1
      Contact( "spremenljivke".Korak2 )
      wire#w2
      "Korak2_DB"(reset := "spremenljivke".reset_DB, finnished => #korak2_finnished)
   END_RUNG
   RUNG wire#w1
      Contact( "spremenljivke".reset_DB )
   END_RUNG wire#w2
   RUNG wire#powerrail
      Contact( "spremenljivke".avtomatično )
      Contact( #korak2_finnished )
      R_Coil( "spremenljivke".Korak2 )
      S_Coil( "spremenljivke".Korak3 )
   END_RUNG
   // the same network as SCL:
   IF "spremenljivke".avtomatično AND ("spremenljivke".Korak2 OR "spremenljivke".reset_DB) THEN
       "Korak2_DB"(reset := "spremenljivke".reset_DB, finnished => #korak2_finnished);   // "Korak2"
   END_IF;
   IF "spremenljivke".avtomatično AND #korak2_finnished THEN
       "spremenljivke".Korak2 := FALSE;
       "spremenljivke".Korak3 := TRUE;
   END_IF;
END_REGION

REGION Network 5
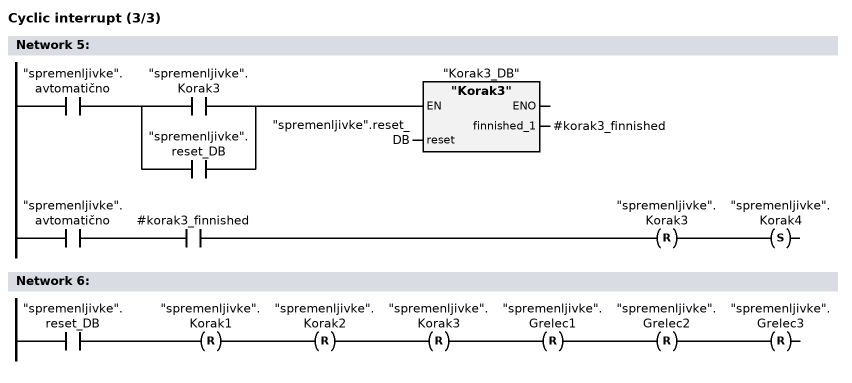
   RUNG wire#powerrail
      Contact( "spremenljivke".avtomatično )
      wire#w1
      Contact( "spremenljivke".Korak3 )
      wire#w2
      "Korak3_DB"(reset := "spremenljivke".reset_DB, finnished_1 => #korak3_finnished)
   END_RUNG
   RUNG wire#w1
      Contact( "spremenljivke".reset_DB )
   END_RUNG wire#w2
   RUNG wire#powerrail
      Contact( "spremenljivke".avtomatično )
      Contact( #korak3_finnished )
      R_Coil( "spremenljivke".Korak3 )
      S_Coil( "spremenljivke".Korak4 )
   END_RUNG
   // the same network as SCL:
   IF "spremenljivke".avtomatično AND ("spremenljivke".Korak3 OR "spremenljivke".reset_DB) THEN
       "Korak3_DB"(reset := "spremenljivke".reset_DB, finnished_1 => #korak3_finnished);   // "Korak3"
   END_IF;
   IF "spremenljivke".avtomatično AND #korak3_finnished THEN
       "spremenljivke".Korak3 := FALSE;
       "spremenljivke".Korak4 := TRUE;
   END_IF;
END_REGION

REGION Network 6
   RUNG wire#powerrail
      Contact( "spremenljivke".reset_DB )
      R_Coil( "spremenljivke".Korak1 )
      R_Coil( "spremenljivke".Korak2 )
      R_Coil( "spremenljivke".Korak3 )
      R_Coil( "spremenljivke".Grelec1 )
      R_Coil( "spremenljivke".Grelec2 )
      R_Coil( "spremenljivke".Grelec3 )
   END_RUNG
   // the same network as SCL:
   IF "spremenljivke".reset_DB THEN
       "spremenljivke".Korak1 := FALSE;
       "spremenljivke".Korak2 := FALSE;
       "spremenljivke".Korak3 := FALSE;
       "spremenljivke".Grelec1 := FALSE;
       "spremenljivke".Grelec2 := FALSE;
       "spremenljivke".Grelec3 := FALSE;
   END_IF;
END_REGION
END_ORGANIZATION_BLOCK

(* ===== HMI "HMI_RT_1" =====
system functions are stored by id; their names below are inferred from use
connection "HMI_Connection_1": ETHERNET, S7_1200_OMS

HMI tags "Default tag table"
   "spremenljivke_reset_DB" : Bool = PLC spremenljivke.reset_DB, 100 ms
   "spremenljivke_Pretok_Voda" : Real = PLC spremenljivke.Pretok_Voda, 1 s
   "spremenljivke_Pretok_alkohol" : Real = PLC spremenljivke.Pretok_alkohol, 1 s
   "spremenljivke_Ventil_alkohol" : Bool = PLC spremenljivke.Ventil_alkohol, 1 s
   "spremenljivke_Ventil_voda" : Bool = PLC spremenljivke.Ventil_voda, 1 s
   "spremenljivke_Pretok_alkohol_mapped" : Real = PLC spremenljivke.Pretok_alkohol_mapped, 1 s
   "spremenljivke_Pretok_Voda_mapped" : Real = PLC spremenljivke.Pretok_Voda_mapped, 1 s
   "spremenljivke_Volumen" : Real = PLC spremenljivke.Volumen, 1 s
   "spremenljivke_%_trenutni" : Real = PLC spremenljivke.%_trenutni, 1 s
   "spremenljivke_Korak1" : Bool = PLC spremenljivke.Korak1, 1 s
   "spremenljivke_Korak2" : Bool = PLC spremenljivke.Korak2, 1 s
   "spremenljivke_Korak3" : Bool = PLC spremenljivke.Korak3, 1 s
   "spremenljivke_Korak4" : Bool = PLC spremenljivke.Korak4, 1 s
   "podatki_procesa_V_žel" : Real = PLC podatki_procesa.V_žel, 1 s
   "podatki_procesa_%_žel" : Real = PLC podatki_procesa.%_žel, 1 s
   "spremenljivke_avtomatično" : Bool = PLC spremenljivke.avtomatično, 1 s
   "spremenljivke_Temperatura" : Real = PLC spremenljivke.Temperatura, 1 s
   "spremenljivke_Grelec1" : Bool = PLC spremenljivke.Grelec1, 1 s
   "spremenljivke_Grelec2" : Bool = PLC spremenljivke.Grelec2, 1 s
   "spremenljivke_Grelec3" : Bool = PLC spremenljivke.Grelec3, 1 s
   "spremenljivke_Mešalo" : Bool = PLC spremenljivke.Mešalo, 1 s
   "podatki_procesa_T_Žel" : Real = PLC podatki_procesa.T_Žel, 1 s
   "spremenljivke_L_sp" : Bool = PLC spremenljivke.L_sp, 1 s
   "spremenljivke_L_zg" : Bool = PLC spremenljivke.L_zg, 1 s
   "spremenljivke_Error" : Word = PLC spremenljivke.Error, 1 s
   "spremenljivke_Ventil_out" : Bool = PLC spremenljivke.Ventil_out, 1 s
   "spremenljivke_glavno_stikalo_DB" : Bool = PLC spremenljivke.glavno_stikalo_DB, 1 s
   "spremenljivke_zasilni_izklop_DB" : Bool = PLC spremenljivke.zasilni_izklop_DB, 1 s
   "spremenljivke_RMSE_T" : Real = PLC spremenljivke.RMSE_T, 1 s

screen "Root screen" 800x480, template "Template_1"
   Button "Button_2" at 20,419 size 70x29; TextOff 'reset'
      on Press: function_b14e0dd5("spremenljivke_reset_DB", 0)
   Button "Button_1" at 646,419 size 96x32; TextOff 'Ročno'
      on Click: ActivateScreen("Ročni_način", 0); ResetBit("spremenljivke_avtomatično")
   GraphicIOField "PlotLight_Round_G" at 727,57 size 25x25; PictureOn "PilotLight_Round_G_On_256c"; PictureOff "PilotLight_Round_G_Off_256c"
      ProcessValue <- "spremenljivke_Korak1"
   GraphicIOField "PlotLight_Round_G_1" at 727,82 size 25x25; PictureOn "PilotLight_Round_G_On_256c"; PictureOff "PilotLight_Round_G_Off_256c"
      ProcessValue <- "spremenljivke_Korak2"
   GraphicIOField "PlotLight_Round_G_2" at 727,107 size 25x25; PictureOn "PilotLight_Round_G_On_256c"; PictureOff "PilotLight_Round_G_Off_256c"
      ProcessValue <- "spremenljivke_Korak3"
   GraphicIOField "PlotLight_Round_G_3" at 727,132 size 25x25; PictureOn "PilotLight_Round_G_On_256c"; PictureOff "PilotLight_Round_G_Off_256c"
      ProcessValue <- "spremenljivke_Korak4"
   IOField "I/O field_1" at 45,59 size 96x32; FormatPattern s999999999.999
      ProcessValue <- "podatki_procesa_V_žel"
   IOField "I/O field_2" at 209,59 size 96x32; FormatPattern s999999999.999
      ProcessValue <- "podatki_procesa_%_žel"
   TextField "Text field_1" at 40,39 size 115x20; Text 'Željen volumen'
   TextField "Text field_2" at 179,40 size 164x20; Text 'Željena koncentracija'
   Button "Button_3" at 530,120 size 96x32; TextOff 'START'
      on Click: SetBit("spremenljivke_Korak1")
   TextField "Text field_3" at 665,60 size 56x20; Text 'Korak1'
   TextField "Text field_4" at 665,86 size 56x20; Text 'Korak2'
   TextField "Text field_5" at 665,110 size 56x20; Text 'Korak3'
   TextField "Text field_6" at 665,133 size 56x20; Text 'Korak4'
   IOField "I/O field_3" at 45,118 size 96x32; FormatPattern s999999999.999
      ProcessValue <- "spremenljivke_Volumen"
   IOField "I/O field_4" at 209,118 size 96x32; FormatPattern s999999999.999
      ProcessValue <- "spremenljivke_%_trenutni"
   TextField "Text field_7" at 32,94 size 134x20; Text 'Trenutni Volumen'
   TextField "Text field_8" at 182,94 size 178x20; Text 'Trenutna koncentracija'
   IOField "I/O field_5" at 366,118 size 96x32; FormatPattern s999999999.999
      ProcessValue <- "spremenljivke_Temperatura"
   IOField "I/O field_6" at 366,62 size 96x32; FormatPattern s999999999.999
      ProcessValue <- "podatki_procesa_T_Žel"
   TextField "Text field_9" at 337,43 size 158x20; Text 'Željena Temperatura'
   TextField "Text field_10" at 338,94 size 172x20; Text 'Trenutna Temperatura'
   GraphicIOField "PlotLight_Round_G_4" at 12,294 size 30x30; PictureOn "PilotLight_Round_G_On_256c"; PictureOff "PilotLight_Round_G_Off_256c"
      ProcessValue <- "spremenljivke_L_sp"
   TextField "Text field_11" at 12,274 size 39x20; Text 'L_sp'
   GraphicIOField "PlotLight_Round_G_5" at 68,294 size 30x30; PictureOff "PilotLight_Round_G_Off_256c"; PictureOn "PilotLight_Round_G_On_256c"
      ProcessValue <- "spremenljivke_L_zg"
   TextField "Text field_12" at 65,274 size 39x20; Text 'L_zg'
   Group "D3_Display_1" at 182,400 size 100x66; Picture "Design_3_NumDisplay_Frame_Small"; FormatPattern 9999
   TextField "Text field_13" at 206,377 size 63x20; Text 'Napake'
   IOField "I/O field_7" at 367,169 size 96x32; FormatPattern 9999999
   TextField "Text field_14" at 342,148 size 177x20; Text 'Temperaturni pogrešek'
   GraphicIOField "PlotLight_Round_G_6" at 424,210 size 30x30; PictureOff "PilotLight_Round_G_Off_256c"; PictureOn "PilotLight_Round_G_On_256c"
      ProcessValue <- "spremenljivke_Grelec1"
   GraphicIOField "PlotLight_Round_G_9" at 424,240 size 30x30; PictureOn "PilotLight_Round_G_On_256c"; PictureOff "PilotLight_Round_G_Off_256c"
      ProcessValue <- "spremenljivke_Grelec2"
   GraphicIOField "PlotLight_Round_G_10" at 424,271 size 30x30; PictureOn "PilotLight_Round_G_On_256c"; PictureOff "PilotLight_Round_G_Off_256c"
      ProcessValue <- "spremenljivke_Grelec3"
   TextField "Text field_15" at 366,214 size 65x20; Text 'Grelec 1'
   TextField "Text field_16" at 367,243 size 65x20; Text 'Grelec 2'
   TextField "Text field_17" at 367,275 size 65x20; Text 'Grelec 3'
   Switch "Toggle_Horizontal_G" at 224,217 size 60x38; CaptionText 'Switch'; TextOff '0'; TextOn '1'; PictureOff "Toggle_Horizontal_G_Off_256c"; PictureOn "Toggle_Horizontal_G_On_256c"
      ProcessValue <- "spremenljivke_Mešalo"
   TextField "Text field_18" at 228,194 size 56x20; Text 'Mešalo'
   GraphicIOField "PlotLight_Round_G_11" at 99,157 size 30x30; PictureOff "PilotLight_Round_G_Off_256c"; PictureOn "PilotLight_Round_G_On_256c"
      ProcessValue <- "spremenljivke_Ventil_alkohol"
   GraphicIOField "PlotLight_Round_G_14" at 99,216 size 30x30; PictureOff "PilotLight_Round_G_Off_256c"; PictureOn "PilotLight_Round_G_On_256c"
      ProcessValue <- "spremenljivke_Ventil_out"
   GraphicIOField "PlotLight_Round_G_15" at 99,186 size 30x30; PictureOff "PilotLight_Round_G_Off_256c"; PictureOn "PilotLight_Round_G_On_256c"
      ProcessValue <- "spremenljivke_Ventil_voda"
   TextField "Text field_19" at 5,162 size 105x20; Text 'Ventil alkohol'
   TextField "Text field_20" at 12,190 size 89x20; Text 'Ventil voda'
   TextField "Text field_21" at 12,220 size 92x20; Text 'Ventil izhod'
   GraphicIOField "PlotLight_Round_G_12" at 239,162 size 30x30; PictureOn "PilotLight_Round_G_On_256c"; PictureOff "PilotLight_Round_G_Off_256c"
      ProcessValue <- "spremenljivke_Mešalo"
   Switch "Pushbutton_Emergency" at 551,249 size 52x52; CaptionText 'Switch'; TextOff '0'; TextOn '1'; PictureOff "Pushbutton_Emergency_Off_256c"; PictureOn "Pushbutton_Emergency_On_256c"
      ProcessValue <- "spremenljivke_zasilni_izklop_DB"
   Switch "Pushbutton_Stop" at 552,174 size 51x52; CaptionText 'Switch'; TextOff '0'; TextOn '1'; PictureOff "Pushbutton_Stop_Off_256c"; PictureOn "Pushbutton_Stop_On_256c"
   Switch "Rotary_RG" at 551,57 size 52x52; CaptionText 'Switch'; TextOff '0'; TextOn '1'; PictureOff "Rotary_RG_Off_256c"; PictureOn "Rotary_RG_On_256c"
      ProcessValue <- "spremenljivke_glavno_stikalo_DB"
   IOField "I/O field_8" at 367,419 size 96x32; FormatPattern s999999999.999
      ProcessValue <- "spremenljivke_RMSE_T"
   TextField "Text field_22" at 343,397 size 150x20; Text 'RMSE TEMPERATURE'
   TextField "Text field_23" at 533,226 size 98x20; Text 'Zasilni izklop'
   TextField "Text field_24" at 559,152 size 39x20; Text 'Stop'
   TextField "Text field_25" at 530,37 size 108x20; Text 'Glavno stikalo'
   GraphicView "D3_NumDisplay_Frame_Small_1" at 182,400 size 100x66; Picture "Design_3_NumDisplay_Frame_Small"
   IOField "D3_I/O field_1" at 182,400 size 100x33; FormatPattern 99999
      ProcessValue <- "spremenljivke_Error"
   TextField "D3_Text field_1" at 182,433 size 100x33; Text '[hPa]'

screen "Ročni_način" 800x480
   Button "Button_1" at 45,76 size 96x32; TextOff 'Ventil Voda'
      on Click: InvertBit("spremenljivke_Ventil_voda")
   Button "Button_2" at 45,31 size 96x32; TextOff 'Ventil Alkohol'
      on Click: InvertBit("spremenljivke_Ventil_alkohol")
   IOField "I/O field_1" at 169,31 size 96x32; FormatPattern s999999999.999
      ProcessValue <- "spremenljivke_Pretok_alkohol_mapped"
   IOField "I/O field_2" at 169,76 size 96x32; FormatPattern s999999999.999
      ProcessValue <- "spremenljivke_Pretok_Voda_mapped"
   Button "Button_3" at 664,422 size 96x32; TextOff 'Avtomatično'
      on Click: ActivateScreen("Root screen", 0); SetBit("spremenljivke_avtomatično")
   IOField "I/O field_3" at 559,51 size 96x32; FormatPattern s999999999.999
      ProcessValue <- "spremenljivke_Volumen"
   IOField "I/O field_4" at 664,51 size 96x32; FormatPattern s999999999.999
      ProcessValue <- "spremenljivke_%_trenutni"
   Button "Button_4" at 45,178 size 96x32; TextOff 'Grelec 1'
      on Click: InvertBit("spremenljivke_Grelec1")
   GraphicIOField "PlotLight_Round_G" at 9,31 size 32x32; PictureOn "PilotLight_Round_G_On_256c"; PictureOff "PilotLight_Round_G_Off_256c"
      ProcessValue <- "spremenljivke_Ventil_alkohol"
   GraphicIOField "PlotLight_Round_G_1" at 9,76 size 32x32; PictureOff "PilotLight_Round_G_Off_256c"; PictureOn "PilotLight_Round_G_On_256c"
      ProcessValue <- "spremenljivke_Ventil_voda"
   Button "Button_5" at 45,220 size 96x32; TextOff 'Grelec 2'
      on Click: InvertBit("spremenljivke_Grelec2")
   Button "Button_6" at 45,259 size 96x32; TextOff 'Grelec 3'
      on Click: InvertBit("spremenljivke_Grelec3")
   GraphicIOField "PlotLight_Round_G_2" at 9,178 size 32x32; PictureOn "PilotLight_Round_G_On_256c"; PictureOff "PilotLight_Round_G_Off_256c"
      ProcessValue <- "spremenljivke_Grelec1"
   GraphicIOField "PlotLight_Round_G_3" at 9,220 size 32x32; PictureOff "PilotLight_Round_G_Off_256c"; PictureOn "PilotLight_Round_G_On_256c"
      ProcessValue <- "spremenljivke_Grelec2"
   GraphicIOField "PlotLight_Round_G_4" at 9,262 size 32x32; PictureOff "PilotLight_Round_G_Off_256c"; PictureOn "PilotLight_Round_G_On_256c"
      ProcessValue <- "spremenljivke_Grelec3"
   IOField "I/O field_5" at 165,220 size 96x32; FormatPattern s999999999.999
      ProcessValue <- "spremenljivke_Temperatura"
   TextField "Text field_1" at 165,190 size 100x20; Text 'Temperatura'
   Button "Button_7" at 45,339 size 96x32; TextOff 'Mešalo'
      on Click: InvertBit("spremenljivke_Mešalo")
   GraphicIOField "PlotLight_Round_G_5" at 9,339 size 32x32; PictureOn "PilotLight_Round_G_On_256c"; PictureOff "PilotLight_Round_G_Off_256c"
      ProcessValue <- "spremenljivke_Mešalo"
*)